// SIMATIC S7-200 SMART project (STEP 7-Micro/WIN SMART), CPU CR40

SYMBOL_TABLE 系统符号
Always_On        SM0.0    // 始终接通
END_SYMBOL_TABLE

ORGANIZATION_BLOCK MAIN:OB1
TITLE=程序注释
BEGIN
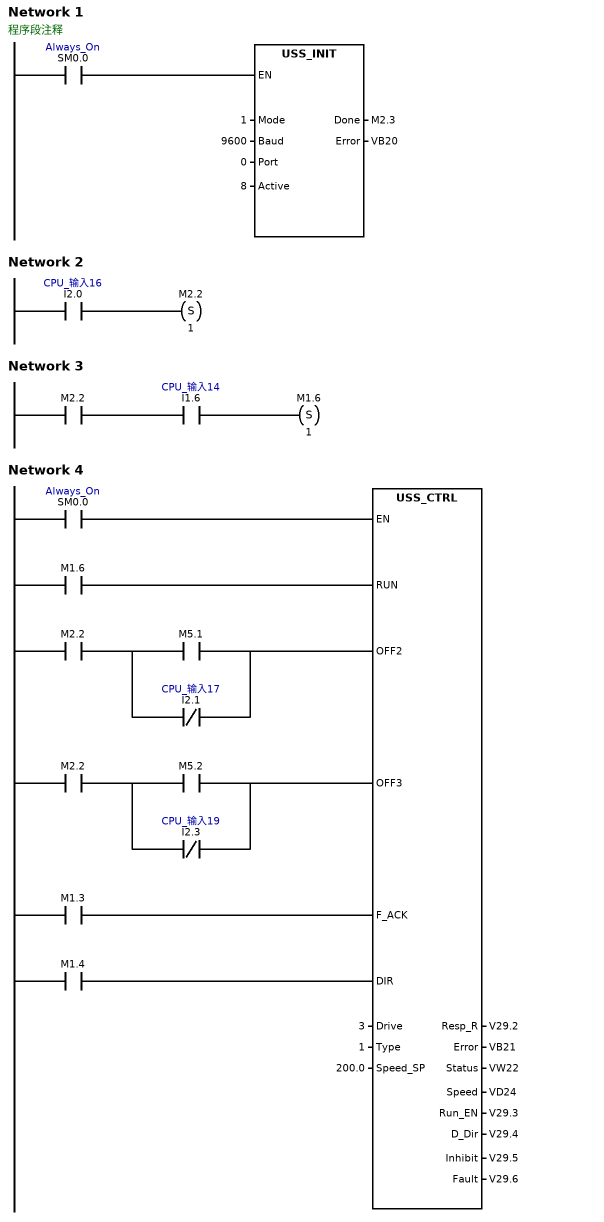
Network 1
// 程序段注释
LD     Always_On:SM0.0
CALL   USS_INIT:SBR1, 1, 9600, 0, 8, M2.3, VB20
Network 2
LD     CPU_输入16:I2.0
S      M2.2, 1
Network 3
LD     M2.2
A      CPU_输入14:I1.6
S      M1.6, 1
Network 4
LD     Always_On:SM0.0
=      L60.0
LD     M1.6
=      L63.7
LD     M2.2
LD     M5.1
ON     CPU_输入17:I2.1
ALD
=      L63.6
LD     M2.2
LD     M5.2
ON     CPU_输入19:I2.3
ALD
=      L63.5
LD     M1.3
=      L63.4
LD     M1.4
=      L63.3
LD     L60.0
CALL   USS_CTRL:SBR5, L63.7, L63.6, L63.5, L63.4, L63.3, 3, 1, 200.0, V29.2, VB21, VW22, VD24, V29.3, V29.4, V29.5, V29.6
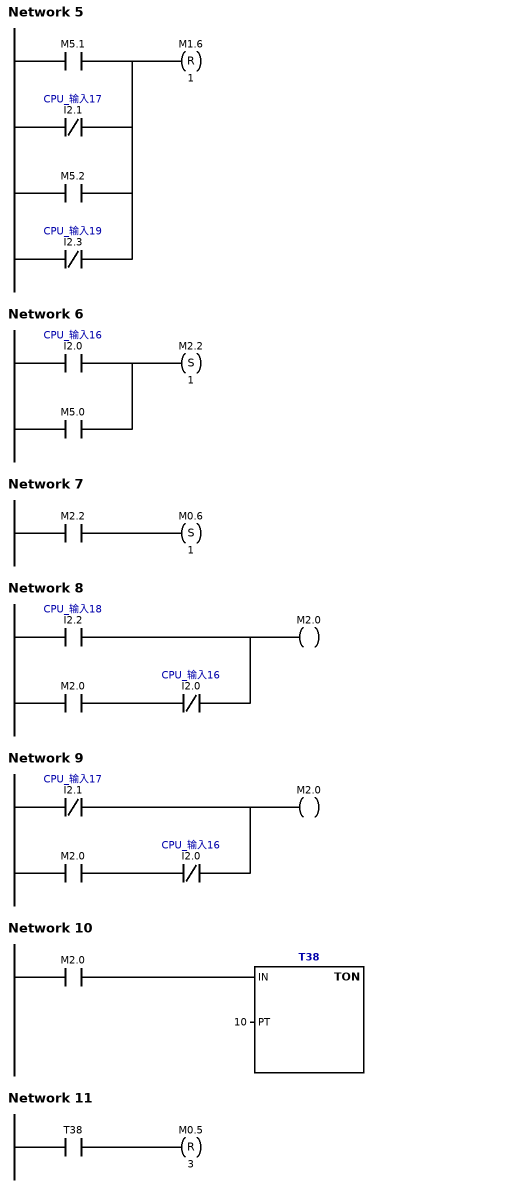
Network 5
LD     M5.1
ON     CPU_输入17:I2.1
O      M5.2
ON     CPU_输入19:I2.3
R      M1.6, 1
Network 6
LD     CPU_输入16:I2.0
O      M5.0
S      M2.2, 1
Network 7
LD     M2.2
S      M0.6, 1
Network 8
LD     CPU_输入18:I2.2
LD     M2.0
AN     CPU_输入16:I2.0
OLD
=      M2.0
Network 9
LDN    CPU_输入17:I2.1
LD     M2.0
AN     CPU_输入16:I2.0
OLD
=      M2.0
Network 10
LD     M2.0
TON    T38, 10
Network 11
LD     T38
R      M0.5, 3
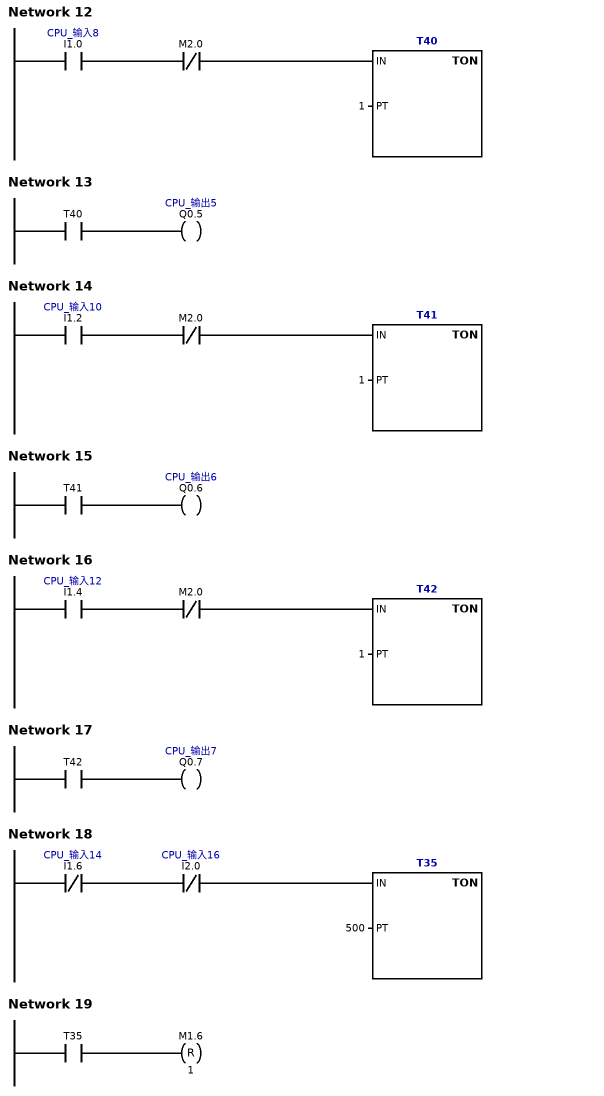
Network 12
LD     CPU_输入8:I1.0
AN     M2.0
TON    T40, 1
Network 13
LD     T40
=      CPU_输出5:Q0.5
Network 14
LD     CPU_输入10:I1.2
AN     M2.0
TON    T41, 1
Network 15
LD     T41
=      CPU_输出6:Q0.6
Network 16
LD     CPU_输入12:I1.4
AN     M2.0
TON    T42, 1
Network 17
LD     T42
=      CPU_输出7:Q0.7
Network 18
LDN    CPU_输入14:I1.6
AN     CPU_输入16:I2.0
TON    T35, 500
Network 19
LD     T35
R      M1.6, 1
END_ORGANIZATION_BLOCK

// SBR1: protected block, not included

// SBR2: protected block, not included

// SBR3: protected block, not included

// SBR4: protected block, not included

// SBR5: protected block, not included

// INT1: protected block, not included
